// TwinCAT 3 PLC project Main
// ProgramVersion: 3.1.4024.0
// libraries:
//   Tc2_Math, * (Beckhoff Automation GmbH)
//   Tc2_Standard, * (Beckhoff Automation GmbH)
//   Tc2_System, * (Beckhoff Automation GmbH)
//   Tc3_Module, * (Beckhoff Automation GmbH)
// project tree:
//   / GlobalTextList.TcGTLO, PlcTask.TcTTO, Visualization Manager.TcVMO (not stored)
//   POUs/ MAIN.TcPOU, PwmSignal.TcPOU, SinusFunction.TcPOU, SquareSignal.TcPOU
//   VISUs/ Visualization.TcVIS
// real-time tasks:
//   TASK PlcTask: cycle T#10ms, priority 20, ADS port 350
//   TASK PlcTask1: cycle T#10ms, priority 21, ADS port 351

CONFIGURATION Main
    RESOURCE PLC ON TwinCAT3
        TASK PlcTask(INTERVAL := T#10ms, PRIORITY := 21);
        PROGRAM MAIN WITH PlcTask : MAIN;
    END_RESOURCE
END_CONFIGURATION

// ---- POUs/MAIN.TcPOU
PROGRAM MAIN
VAR
	SinusValue :	REAL := 0;
	SquareValue:	REAL := 0;
	PWMValue:		REAL := 0;
	t:				REAL := 0;
END_VAR

SinusValue := SinusFunction(A:=2,yoff:=0,w:=2,t:=t);
SquareValue := SquareSignal(ymin:= 4, ymax := 3, w:= 5, yoff:= -1, t:=t);
PWMValue := PwmSignal(ymin:= 4, ymax := 3, w:= 5, yoff:= -1, t:=t, PWM:= 0.7);

t := t + 0.01;

END_PROGRAM

// ---- POUs/SinusFunction.TcPOU
FUNCTION SinusFunction : REAL
VAR_INPUT
	A : 	REAL; 		//Amplitude
	yoff : 	REAL;		//Offset
	w : 	REAL;		//Kreisfrequenz
	t : 	REAL;		//Zeit
END_VAR
VAR
END_VAR

SinusFunction := A * sin(w*t) + yoff;
RETURN;

END_FUNCTION

// ---- POUs/SquareSignal.TcPOU
FUNCTION SquareSignal : REAL
VAR_INPUT
	ymin:				REAL; 	//Minimalwert
	ymax:				REAL; 	//Maximalwert
	w:					REAL; 	//Kreisfrequenz
	yoff:				REAL; 	//yoffset
	t : 				REAL;	//Zeit
END_VAR
VAR
	tempTime:			REAL;
	tempVar:			INT;
END_VAR

tempTime := LMOD(lr_Value:=t,lr_Arg:=(2*PI)/w)/((2*PI)/w);

IF(tempTime >= (0.5)) THEN
	SquareSignal := ymax + yoff;
	RETURN;
ELSE
	SquareSignal := ymin + yoff;
	RETURN;
END_IF

END_FUNCTION

// ---- POUs/PwmSignal.TcPOU
FUNCTION PwmSignal : REAL
VAR_INPUT
	ymin:				REAL; 	//Minimalwert
	ymax:				REAL; 	//Maximalwert
	w:					REAL; 	//Kreisfrequenz
	yoff:				REAL; 	//yoffset
	PWM:				REAL;	//PWM 0.0 ... 1.0%
	t : 				REAL;	//Zeit
END_VAR
VAR
	tempTime:			REAL;
END_VAR

tempTime := LMOD(lr_Value:=t,lr_Arg:=(2*PI)/w)/((2*PI)/w);

IF(PWM = 1) THEN
	PwmSignal := ymax + yoff;
	RETURN;
END_IF
IF(tempTime <= (1-PWM)) THEN
	PwmSignal := ymin + yoff;
	RETURN;
ELSE
	PwmSignal := ymax + yoff;
	RETURN;
END_IF

END_FUNCTION

// ---- VISUs/Visualization.TcVIS
VISUALIZATION Visualization  // 2x2
END_VISUALIZATION
